TYPE udt_AdsAddr :
STRUCT
(*Used to read in the ADS address of the AX5805*)
(*Data structure must remain in this order*)
	netId:		ARRAY [0..5] OF USINT;
END_STRUCT
END_TYPE

(* stored: Version 1.1.0.1, ProductVersion 3.1.4024.9
   DUT udt_AdsAddr: Id {16437dac-49e9-4057-bd6f-0b30564038b3} *)
